// TIA Portal project "assemblerProject" (V17)
// Vorlageprojekt für das Buch mit Zielsystem S7-1200

(* hardware
DEVICE "S7-1200-Station_1"  S7-1200 Station
   slot 0: "Baugruppenträger_0"  Rack  V1.0
   slot 1: "PLC_1"  CPU 1211C DC/DC/DC  6ES7 211-1AE40-0XB0  V4.1
*)

// ===== PLC "PLC_1"  CPU 1211C DC/DC/DC =====

VAR_GLOBAL   // PLC tag table "inputs"
   "moving x" AT %I0.0 : Bool;
   "moving z" AT %I0.1 : Bool;
   "item detected" AT %I0.2 : Bool;
   "lid at place" AT %I0.3 : Bool;
   "lid clamped" AT %I0.4 : Bool;
   "pos. at limit (lids)" AT %I0.5 : Bool;
   "base at place" AT %I0.6 : Bool;
   "base clamped" AT %I0.7 : Bool;
   "pos. at limit (base)" AT %I1.0 : Bool;
   "part leaving" AT %I1.1 : Bool;
   "start PB" AT %I1.2 : Bool;
   "reset" AT %I1.3 : Bool;
   "stop PB" AT %I1.4 : Bool;
   "emergency stop PB" AT %I1.5 : Bool;
   "auto" AT %I1.6 : Bool;
   "item grabbed" AT %I1.7 : Bool;
   "item leaving" AT %M3.5 : Bool;
END_VAR

VAR_GLOBAL   // PLC tag table "outputs"
   "move x" AT %Q0.0 : Bool;
   "move z" AT %Q0.1 : Bool;
   "grab" AT %Q0.2 : Bool;
   "lids conveyor" AT %Q0.3 : Bool;
   "clamp lid" AT %Q0.4 : Bool;
   "pos. raise (lids)" AT %Q0.5 : Bool;
   "base conveyor" AT %Q0.6 : Bool;
   "clamp base" AT %Q0.7 : Bool;
   "pos. raise (base)" AT %Q1.0 : Bool;
   "start light" AT %Q1.1 : Bool;
   "reset light" AT %Q1.2 : Bool;
   "stop light" AT %Q1.3 : Bool;
   "counter" AT %QW30 : Int;
END_VAR

VAR_GLOBAL   // PLC tag table "memories"
   "activate" AT %M0.0 : Bool;
   "sequence" AT %MW1 : Int;
   "conveyor run" AT %M0.1 : Bool;
   "clamp activate" AT %M0.2 : Bool;
   "lid place" AT %M0.3 : Bool;
   "base place" AT %M0.4 : Bool;
   "moving x sensor" AT %M0.5 : Bool;
   "grab activate" AT %M0.6 : Bool;
   "moving z lid activate" AT %M0.7 : Bool;
   "moving x activate" AT %M3.0 : Bool;
   "moving z base activate" AT %M3.1 : Bool;
   "reset process" AT %M3.2 : Bool;
   "pos. activate" AT %M3.3 : Bool;
   "items exit" AT %M3.4 : Bool;
   "process reset" AT %M3.6 : Bool;
   "moving z lid release" AT %M3.7 : Bool;
   "moving z base neew" AT %M4.0 : Bool;
   "grab release" AT %M4.1 : Bool;
   "release x and z move" AT %M4.2 : Bool;
   "close pos." AT %M4.3 : Bool;
   "part leave" AT %M4.4 : Bool;
END_VAR

DATA_BLOCK "cell zone 1 sequencer"   // DB6
{ S7_Optimized_Access := 'TRUE' }
VERSION : 0.1
// stored: InstanceOfName 00 sequencer
"00 sequencer"
BEGIN
END_DATA_BLOCK

DATA_BLOCK "cell zone 1 output"   // DB8
{ S7_Optimized_Access := 'TRUE' }
VERSION : 0.1
// stored: InstanceOfName 01 output
"01 output"
BEGIN
END_DATA_BLOCK

// folder: System blocks/Program resources

DATA_BLOCK "IEC_Timer_0_DB"   // DB1
{ S7_Optimized_Access := 'TRUE' }
AUTHOR : Simatic
FAMILY : IEC
NAME : IEC_TMR
VERSION : 1.0
// stored: InstanceOfName IEC_TIMER
"IEC_TIMER"
BEGIN
END_DATA_BLOCK

DATA_BLOCK "IEC_Timer_0_DB_1"   // DB2
{ S7_Optimized_Access := 'TRUE' }
AUTHOR : Simatic
FAMILY : IEC
NAME : IEC_TMR
VERSION : 1.0
// stored: InstanceOfName IEC_TIMER
"IEC_TIMER"
BEGIN
END_DATA_BLOCK

DATA_BLOCK "IEC_Timer_0_DB_2"   // DB3
{ S7_Optimized_Access := 'TRUE' }
AUTHOR : Simatic
FAMILY : IEC
NAME : IEC_TMR
VERSION : 1.0
// stored: InstanceOfName IEC_TIMER
"IEC_TIMER"
BEGIN
END_DATA_BLOCK

DATA_BLOCK "IEC_Timer_0_DB_3"   // DB4
{ S7_Optimized_Access := 'TRUE' }
AUTHOR : Simatic
FAMILY : IEC
NAME : IEC_TMR
VERSION : 1.0
// stored: InstanceOfName IEC_TIMER
"IEC_TIMER"
BEGIN
END_DATA_BLOCK

DATA_BLOCK "IEC_Timer_0_DB_4"   // DB5
{ S7_Optimized_Access := 'TRUE' }
AUTHOR : Simatic
FAMILY : IEC
NAME : IEC_TMR
VERSION : 1.0
// stored: InstanceOfName IEC_TIMER
"IEC_TIMER"
BEGIN
END_DATA_BLOCK

DATA_BLOCK "IEC_Counter_0_DB_1"   // DB7
{ S7_Optimized_Access := 'TRUE' }
AUTHOR : Simatic
FAMILY : IEC
NAME : CNTR
VERSION : 1.0
// stored: InstanceOfName IEC_COUNTER
"IEC_COUNTER"
BEGIN
END_DATA_BLOCK

// folder: (top level)

FUNCTION_BLOCK "00 sequencer"   // FB1, LAD
{ S7_Optimized_Access := 'TRUE' }
VERSION : 0.1
   VAR_INPUT
      "moving x" : Bool;
      "moving z" : Bool;
      "item detected" : Bool;
      "lid at place" : Bool;
      "lid clamped" : Bool;
      "pos. at limit (lids)" : Bool;
      "base at place" : Bool;
      "base clamped" : Bool;
      "pos. at limit (base)" : Bool;
      "part leaving" : Bool;
      "start PB" : Bool;
      reset : Bool;
      "stop PB" : Bool;
      "emergency stop PB" : Bool;
      auto : Bool;
      "item grabbed" : Bool;
      "item leaving" : Bool;
   END_VAR
   VAR_OUTPUT
      "move x" : Bool;
      "move z" : Bool;
      grab : Bool;
      "lids conveyor" : Bool;
      "clamp lid" : Bool;
      "pos. raise (lids)" : Bool;
      "base conveyor" : Bool;
      "clamp base" : Bool;
      "pos. raise (base)" : Bool;
      "start light" : Bool;
      "reset light" : Bool;
      "stop light" : Bool;
      "counter" : Bool;
   END_VAR
BEGIN

REGION Network 1: step 0: activete process
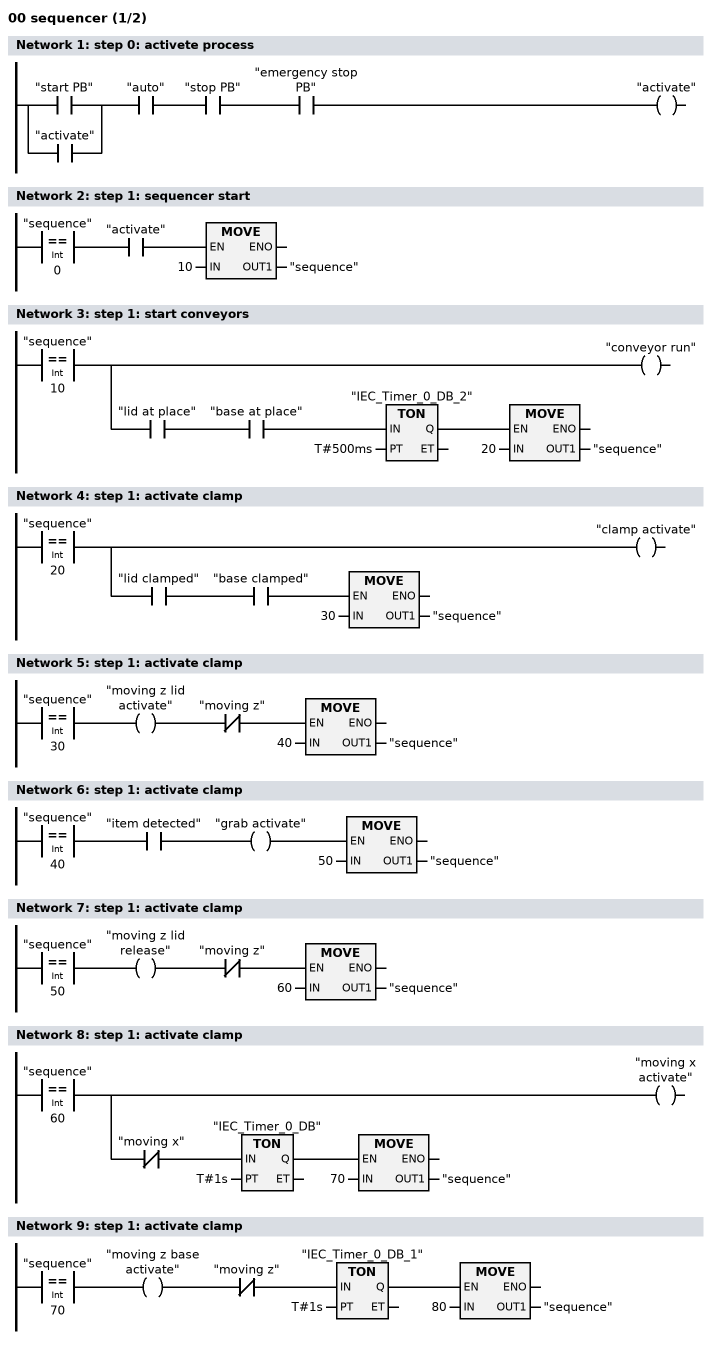
   RUNG wire#powerrail
      Contact( "start PB" )
      wire#w1
      Contact( "auto" )
      Contact( "stop PB" )
      Contact( "emergency stop PB" )
      Coil( "activate" )
   END_RUNG
   RUNG wire#powerrail
      Contact( "activate" )
   END_RUNG wire#w1
   // the same network as SCL:
   "activate" := ("start PB" OR "activate") AND "auto" AND "stop PB" AND "emergency stop PB";
END_REGION

REGION Network 2: step 1: sequencer start
   RUNG wire#powerrail
      { S7_Templates := "SrcType := Int" } EQ_Contact(in1 := "sequence", in2 := 0)
      Contact( "activate" )
      Move(in := 10, out1 => "sequence")
   END_RUNG
   // the same network as SCL:
   IF ("sequence" = 0) AND "activate" THEN "sequence" := 10; END_IF;
END_REGION

REGION Network 3: step 1: start conveyors
   "conveyor run" := "sequence" = 10;
   "IEC_Timer_0_DB_2".TON(IN := "conveyor run" AND "lid at place" AND "base at place", PT := T#500ms);
   IF "IEC_Timer_0_DB_2".Q THEN "sequence" := 20; END_IF;
END_REGION

REGION Network 4: step 1: activate clamp
   RUNG wire#powerrail
      { S7_Templates := "SrcType := Int" } EQ_Contact(in1 := "sequence", in2 := 20)
      wire#w1
      Coil( "clamp activate" )
   END_RUNG
   RUNG wire#w1
      Contact( "lid clamped" )
      Contact( "base clamped" )
      Move(in := 30, out1 => "sequence")
   END_RUNG
   // the same network as SCL:
   "clamp activate" := "sequence" = 20;
   IF "clamp activate" AND "lid clamped" AND "base clamped" THEN "sequence" := 30; END_IF;
END_REGION

REGION Network 5: step 1: activate clamp
   RUNG wire#powerrail
      { S7_Templates := "SrcType := Int" } EQ_Contact(in1 := "sequence", in2 := 30)
      Coil( "moving z lid activate" )
      I_Contact( "moving z" )
      Move(in := 40, out1 => "sequence")
   END_RUNG
   // the same network as SCL:
   "moving z lid activate" := "sequence" = 30;
   IF "moving z lid activate" AND NOT "moving z" THEN "sequence" := 40; END_IF;
END_REGION

REGION Network 6: step 1: activate clamp
   RUNG wire#powerrail
      { S7_Templates := "SrcType := Int" } EQ_Contact(in1 := "sequence", in2 := 40)
      Contact( "item detected" )
      Coil( "grab activate" )
      Move(in := 50, out1 => "sequence")
   END_RUNG
   // the same network as SCL:
   "grab activate" := ("sequence" = 40) AND "item detected";
   IF "grab activate" THEN "sequence" := 50; END_IF;
END_REGION

REGION Network 7: step 1: activate clamp
   RUNG wire#powerrail
      { S7_Templates := "SrcType := Int" } EQ_Contact(in1 := "sequence", in2 := 50)
      Coil( "moving z lid release" )
      I_Contact( "moving z" )
      Move(in := 60, out1 => "sequence")
   END_RUNG
   // the same network as SCL:
   "moving z lid release" := "sequence" = 50;
   IF "moving z lid release" AND NOT "moving z" THEN "sequence" := 60; END_IF;
END_REGION

REGION Network 8: step 1: activate clamp
   "moving x activate" := "sequence" = 60;
   "IEC_Timer_0_DB".TON(IN := "moving x activate" AND NOT "moving x", PT := T#1s);
   IF "IEC_Timer_0_DB".Q THEN "sequence" := 70; END_IF;
END_REGION

REGION Network 9: step 1: activate clamp
   "moving z base activate" := "sequence" = 70;
   "IEC_Timer_0_DB_1".TON(IN := "moving z base activate" AND NOT "moving z", PT := T#1s);
   IF "IEC_Timer_0_DB_1".Q THEN "sequence" := 80; END_IF;
END_REGION

REGION Network 10: step 1: activate clamp
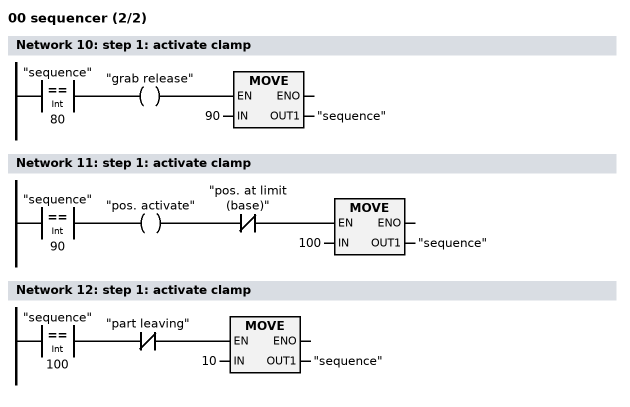
   RUNG wire#powerrail
      { S7_Templates := "SrcType := Int" } EQ_Contact(in1 := "sequence", in2 := 80)
      Coil( "grab release" )
      Move(in := 90, out1 => "sequence")
   END_RUNG
   // the same network as SCL:
   "grab release" := "sequence" = 80;
   IF "grab release" THEN "sequence" := 90; END_IF;
END_REGION

REGION Network 11: step 1: activate clamp
   RUNG wire#powerrail
      { S7_Templates := "SrcType := Int" } EQ_Contact(in1 := "sequence", in2 := 90)
      Coil( "pos. activate" )
      I_Contact( "pos. at limit (base)" )
      Move(in := 100, out1 => "sequence")
   END_RUNG
   // the same network as SCL:
   "pos. activate" := "sequence" = 90;
   IF "pos. activate" AND NOT "pos. at limit (base)" THEN "sequence" := 100; END_IF;
END_REGION

REGION Network 12: step 1: activate clamp
   RUNG wire#powerrail
      { S7_Templates := "SrcType := Int" } EQ_Contact(in1 := "sequence", in2 := 100)
      I_Contact( "part leaving" )
      Move(in := 10, out1 => "sequence")
   END_RUNG
   // the same network as SCL:
   IF ("sequence" = 100) AND NOT "part leaving" THEN "sequence" := 10; END_IF;
END_REGION
END_FUNCTION_BLOCK

FUNCTION_BLOCK "01 output"   // FB2, LAD
{ S7_Optimized_Access := 'TRUE' }
VERSION : 0.1
   VAR_INPUT
      "moving x" : Bool;
      "moving z" : Bool;
      "item detected" : Bool;
      "lid at place" : Bool;
      "lid clamped" : Bool;
      "pos. at limit (lids)" : Bool;
      "base at place" : Bool;
      "base clamped" : Bool;
      "pos. at limit (base)" : Bool;
      "part leaving" : Bool;
      "start PB" : Bool;
      reset : Bool;
      "stop PB" : Bool;
      "emergency stop PB" : Bool;
      auto : Bool;
      "item grabbed" : Bool;
      "item leaving" : Bool;
   END_VAR
   VAR_OUTPUT
      "move x" : Bool;
      "move z" : Bool;
      grab : Bool;
      "lids conveyor" : Bool;
      "clamp lid" : Bool;
      "pos. raise (lids)" : Bool;
      "base conveyor" : Bool;
      "clamp base" : Bool;
      "pos. raise (base)" : Bool;
      "start light" : Bool;
      "reset light" : Bool;
      "stop light" : Bool;
      "counter" : Bool;
   END_VAR
   VAR_TEMP   // added for the SCL form of the ladder/FBD networks
      _w1 : Bool;
   END_VAR
BEGIN

REGION Network 1: start light
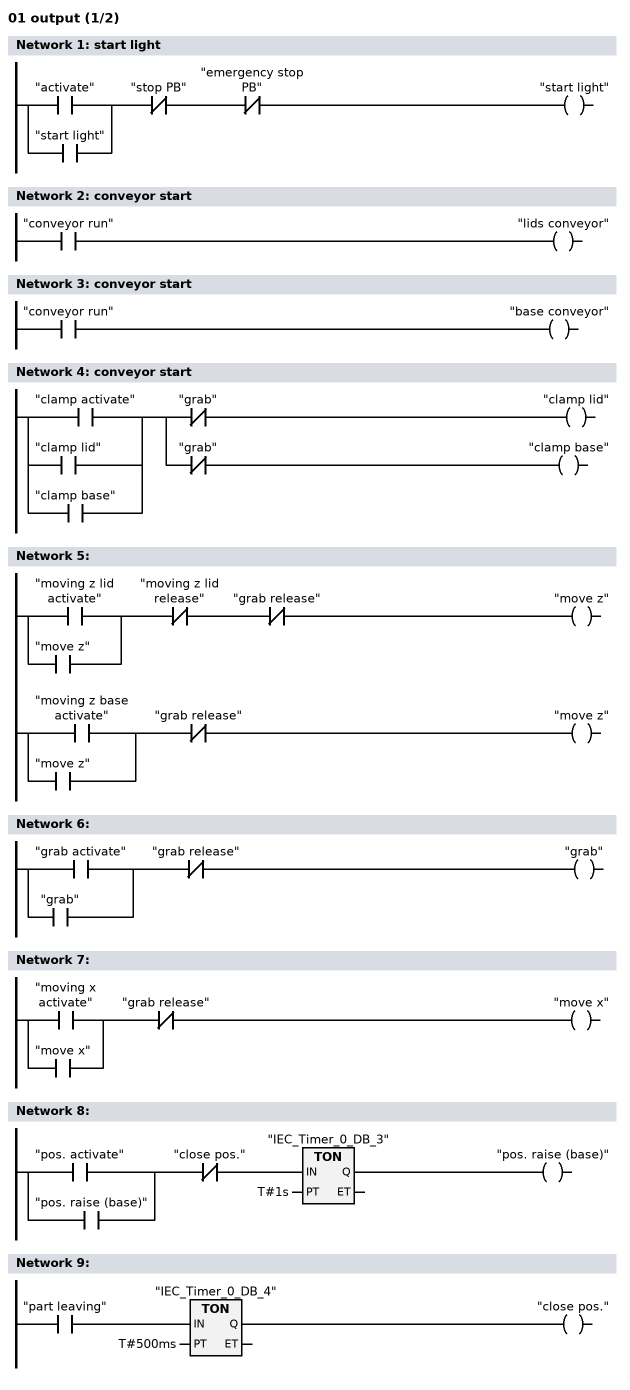
   RUNG wire#powerrail
      Contact( "activate" )
      wire#w1
      I_Contact( "stop PB" )
      I_Contact( "emergency stop PB" )
      Coil( "start light" )
   END_RUNG
   RUNG wire#powerrail
      Contact( "start light" )
   END_RUNG wire#w1
   // the same network as SCL:
   "start light" := ("activate" OR "start light") AND NOT "stop PB" AND NOT "emergency stop PB";
END_REGION

REGION Network 2: conveyor start
   RUNG wire#powerrail
      Contact( "conveyor run" )
      Coil( "lids conveyor" )
   END_RUNG
   // the same network as SCL:
   "lids conveyor" := "conveyor run";
END_REGION

REGION Network 3: conveyor start
   RUNG wire#powerrail
      Contact( "conveyor run" )
      Coil( "base conveyor" )
   END_RUNG
   // the same network as SCL:
   "base conveyor" := "conveyor run";
END_REGION

REGION Network 4: conveyor start
   RUNG wire#powerrail
      Contact( "clamp activate" )
      wire#w1
      I_Contact( "grab" )
      Coil( "clamp lid" )
   END_RUNG
   RUNG wire#powerrail
      Contact( "clamp lid" )
   END_RUNG wire#w1
   RUNG wire#powerrail
      Contact( "clamp base" )
   END_RUNG wire#w1
   RUNG wire#w1
      I_Contact( "grab" )
      Coil( "clamp base" )
   END_RUNG
   // the same network as SCL:
   #_w1 := "clamp activate" OR "clamp lid" OR "clamp base";
   "clamp lid" := #_w1 AND NOT "grab";
   "clamp base" := #_w1 AND NOT "grab";
END_REGION

REGION Network 5
   RUNG wire#powerrail
      Contact( "moving z lid activate" )
      wire#w1
      I_Contact( "moving z lid release" )
      I_Contact( "grab release" )
      Coil( "move z" )
   END_RUNG
   RUNG wire#powerrail
      Contact( "move z" )
   END_RUNG wire#w1
   RUNG wire#powerrail
      Contact( "moving z base activate" )
      wire#w2
      I_Contact( "grab release" )
      Coil( "move z" )
   END_RUNG
   RUNG wire#powerrail
      Contact( "move z" )
   END_RUNG wire#w2
   // the same network as SCL:
   "move z" := ("moving z lid activate" OR "move z") AND NOT "moving z lid release" AND NOT "grab release";
   "move z" := ("moving z base activate" OR "move z") AND NOT "grab release";
END_REGION

REGION Network 6
   RUNG wire#powerrail
      Contact( "grab activate" )
      wire#w1
      I_Contact( "grab release" )
      Coil( "grab" )
   END_RUNG
   RUNG wire#powerrail
      Contact( "grab" )
   END_RUNG wire#w1
   // the same network as SCL:
   "grab" := ("grab activate" OR "grab") AND NOT "grab release";
END_REGION

REGION Network 7
   RUNG wire#powerrail
      Contact( "moving x activate" )
      wire#w1
      I_Contact( "grab release" )
      Coil( "move x" )
   END_RUNG
   RUNG wire#powerrail
      Contact( "move x" )
   END_RUNG wire#w1
   // the same network as SCL:
   "move x" := ("moving x activate" OR "move x") AND NOT "grab release";
END_REGION

REGION Network 8
   "IEC_Timer_0_DB_3".TON(IN := ("pos. activate" OR "pos. raise (base)") AND NOT "close pos.", PT := T#1s);
   "pos. raise (base)" := "IEC_Timer_0_DB_3".Q;
END_REGION

REGION Network 9
   "IEC_Timer_0_DB_4".TON(IN := "part leaving", PT := T#500ms);
   "close pos." := "IEC_Timer_0_DB_4".Q;
END_REGION

REGION Network 10
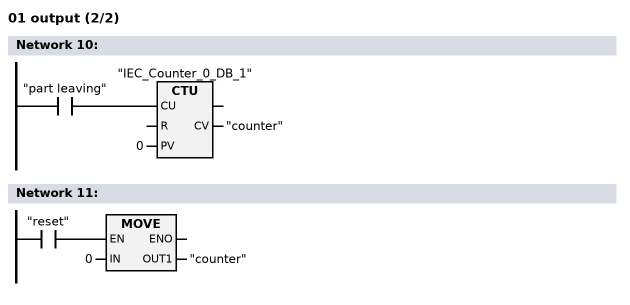
   "IEC_Counter_0_DB_1".CTU(CU := "part leaving", PV := 0, CV => "counter");
END_REGION

REGION Network 11
   RUNG wire#powerrail
      Contact( "reset" )
      Move(in := 0, out1 => "counter")
   END_RUNG
   // the same network as SCL:
   IF "reset" THEN "counter" := 0; END_IF;
END_REGION
END_FUNCTION_BLOCK

FUNCTION "MHJ-PLC-Lab-Function-S71200" : Void   // FC9000, SCL
{ S7_Optimized_Access := 'TRUE' }
VERSION : 0.1
   VAR_TEMP
      rdTimeReturn : Int;
      outputTime : DTL;
      SyncVal : Byte;
      forVal : Int;
      forVal_2 : Int;
      Value : Byte;
   END_VAR
   VAR CONSTANT
      CompVal : Byte := 16#34;
      Value_01 : Byte := 16#11;
      Value_01_DW : DWord := 16#A165_D992;
      Value_02_DW : DWord := 16#58BE_4401;
   END_VAR
BEGIN

   #Value:=PEEK(area := 16#82,
        dbNumber := 0,
        byteOffset := 511);
   #Value := #Value + 1;

   POKE(area := 16#82,
        dbNumber := 0,
        byteOffset := 511,
        value := #Value);

   POKE(area:=16#81,
        dbNumber:=0,
        byteOffset:=1016,
        value:=#Value_01_DW);
   POKE(area := 16#81,
        dbNumber := 0,
        byteOffset := 1020,
        value := #Value_02_DW);

   POKE(area := 16#81,
        dbNumber := 0,
        byteOffset := 511,
        value := B#16#00);

   FOR #forVal := 0 TO 120 DO
       FOR #forVal_2:=0 TO 10 DO
           #rdTimeReturn:=RD_SYS_T(#outputTime);
           #rdTimeReturn := WR_SYS_T(#outputTime);
           #rdTimeReturn := RD_SYS_T(#outputTime);
           #rdTimeReturn := WR_SYS_T(#outputTime);
       END_FOR;
       #SyncVal:= PEEK(area := 16#81,
                      dbNumber := 0,
                      byteOffset := 511);
       IF #SyncVal = #CompVal THEN
          GOTO M_1;
       END_IF;
   END_FOR;
   RETURN;

   M_1:
   POKE(area := 16#81,
        dbNumber := 0,
        byteOffset := 511,
        value := B#16#0);
END_FUNCTION

ORGANIZATION_BLOCK "Main"   // OB1, FBD, ProgramCycle
TITLE = "Main Program Sweep (Cycle)"
{ S7_Optimized_Access := 'TRUE' }
VERSION : 0.1
   VAR_INPUT
      Initial_Call : Bool;   // Initial call of this OB
      Remanence : Bool;   // =True, if remanent data are available
   END_VAR
BEGIN

REGION Network 1: Konnektierungsbaustein für PLC-Lab
   // Im Netzwerk 1 wird der Konnektierungsbaustein für PLC-Lab aufgerufen.
   // Dieser Aufruf darf nicht entfernt werden!
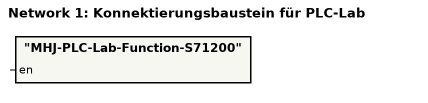
   "MHJ-PLC-Lab-Function-S71200"();
END_REGION

REGION Network 2: Ihr Programm
   // Schreiben Sie ab Netzwerk 2 Ihr Programm
END_REGION
END_ORGANIZATION_BLOCK

ORGANIZATION_BLOCK "sequencer zone 1"   // OB123, FBD, ProgramCycle
TITLE = "Main Program Sweep (Cycle)"
{ S7_Optimized_Access := 'TRUE' }
VERSION : 0.1
   VAR_INPUT
      Initial_Call : Bool;   // Initial call of this OB
      Remanence : Bool;   // =True, if remanent data are available
   END_VAR
BEGIN

REGION Network 1
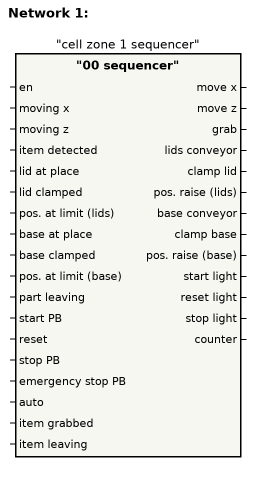
   "cell zone 1 sequencer"();   // "00 sequencer"
END_REGION
END_ORGANIZATION_BLOCK

ORGANIZATION_BLOCK "output zone 1"   // OB124, FBD, ProgramCycle
TITLE = "Main Program Sweep (Cycle)"
{ S7_Optimized_Access := 'TRUE' }
VERSION : 0.1
   VAR_INPUT
      Initial_Call : Bool;   // Initial call of this OB
      Remanence : Bool;   // =True, if remanent data are available
   END_VAR
BEGIN

REGION Network 1
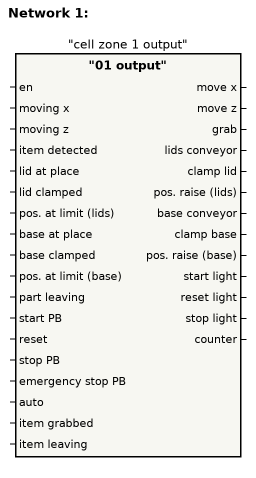
   "cell zone 1 output"();   // "01 output"
END_REGION
END_ORGANIZATION_BLOCK